TYPE E_ActionStatus :
(
	ACTIONSTATUS_Idle := 0,
	ACTIONSTATUS_Active,
	ACTIONSTATUS_PauseRequest,
	ACTIONSTATUS_Pause,
	ACTIONSTATUS_Ready,
	ACTIONSTATUS_Error
)USINT;
END_TYPE

(* stored: Version 1.1.0.1, ProductVersion 3.1.4022.10
   DUT E_ActionStatus: Id {1163c3de-e759-411e-aaee-3971b2596de2} *)
